TYPE ST_AXIS_SETUP_MODE_STATUS :
STRUCT
END_STRUCT
END_TYPE

(* stored: Version 1.1.0.1, ProductVersion 3.1.4024.11
   DUT ST_AXIS_SETUP_MODE_STATUS: Id {3da78e33-4003-4905-becd-390ba288410e} *)
